// TIA Portal V19 export
DATA_BLOCK "FMTemperature Sts"   // DB25
// stored: InstanceOfName FmStsCodes, InstanceOfType FB
"FmStsCodes"
   // VAR_INPUT
   //    StsIn : Byte;
   // END_VAR
   // VAR_OUTPUT
   //    "Maint alarm" : Bool;
   //    "Process Issue" : Bool;
   //    "Function Check" : Bool;
   //    "Uncertain Initial val" : Bool;
   //    "Uncertain Maint demand" : Bool;
   //    "Uncertain Process Related" : Bool;
   //    Ok : Bool;
   //    "OK maint advised" : Bool;
   //    "OK function Check" : Bool;
   // END_VAR
   // VAR
   //    Val1 : Byte;
   // END_VAR
BEGIN
END_DATA_BLOCK
